DATA_BLOCK "AutoProcessDataPopUp_DB"
{ S7_Optimized_Access := 'TRUE' }
VERSION : 0.1
NON_RETAIN
// ATTRIBUTES
// AUTO_NUMBER = True
// BLOCK_NUMBER = 2
// END_ATTRIBUTES
"AutoProcessDataPopUp"

BEGIN

END_DATA_BLOCK

